(********************* G.D S.p.A. - Technical Department ***********************************
This program has been generated automatically from Application Designer DE&F
********************************************************************************************)
PROGRAM dbg_csp_case_openflap_sensors
VAR
  open_flap_ls_di_shd : digital_input_shadow;
  open_flap_ls_di_dchk_shd : check_section_shadow;
  open_flap_os_di_shd : digital_input_shadow;
  open_flap_os_di_dchk_shd : check_section_shadow;
END_VAR

_objects_manager();

IF	g_application_status <> APPLICATION_STATUS_RUNNING
THEN
	RETURN;
END_IF

CASE process_get_mode(CONVERSION_this := dbg_root.prc) OF
	MODE_ABSENT,
	MODE_INACTIVE:
		RETURN;
	MODE_TEST:
		RETURN;
END_CASE

ACTION _objects_manager:
IF	objects_initialization()
THEN
	digital_input_shadow_init(
		sim_mode:= SHADOW_SIMULATION_MODE_AUTOMATIC, 
		father:= csp_case_openflap_sensors.open_flap_ls_di, 
		process:= dbg_root.prc, 
		CONVERSION_this:= open_flap_ls_di_shd);

	check_section_shadow_init(
		sim_mode:= SHADOW_SIMULATION_MODE_AUTOMATIC, 
		father:= csp_case_openflap_sensors.open_major_flap_ls_di_dchk, 
		process:= dbg_root.prc, 
		CONVERSION_this:= open_flap_ls_di_dchk_shd);

	digital_input_shadow_init(
		sim_mode:= SHADOW_SIMULATION_MODE_AUTOMATIC, 
		father:= csp_case_openflap_sensors.open_flap_os_di, 
		process:= dbg_root.prc, 
		CONVERSION_this:= open_flap_os_di_shd);

	check_section_shadow_init(
		sim_mode:= SHADOW_SIMULATION_MODE_AUTOMATIC, 
		father:= csp_case_openflap_sensors.open_major_flap_os_di_dchk, 
		process:= dbg_root.prc, 
		CONVERSION_this:= open_flap_os_di_dchk_shd);

	RETURN;
END_IF

IF	objects_running()
THEN
	digital_input_shadow_cycle(open_flap_ls_di_shd);
	digital_input_shadow_cycle(open_flap_os_di_shd);
END_IF
END_ACTION

END_PROGRAM

(* stored: Version 1.1.0.1, ProductVersion 3.1.4024.3
   POU dbg_csp_case_openflap_sensors: Id {434fac44-e123-44ff-ae0e-de5864246d17}, SpecialFunc None
   Action _objects_manager: Id {ebf17ce7-7d24-4f92-a2db-9342c25bf24d} *)
